INTERFACE I_IterableElementCollection

METHOD createIterator : REFERENCE TO FB_ElementIterator
VAR_INPUT
END_VAR
END_METHOD

END_INTERFACE

(* stored: Version 1.1.0.1
   Itf I_IterableElementCollection: Id {1b1f58f0-94ac-49f1-969c-bd29e8847c8b}
   Method createIterator: Id {05b3aa24-8817-442d-84e9-4ef418fc1650} *)
